// TwinCAT 3 PLC project TrafficPLC
// ProgramVersion: 3.1.4024.0
// libraries:
//   Tc2_Standard, * (Beckhoff Automation GmbH)
//   Tc2_System, * (Beckhoff Automation GmbH)
//   Tc3_Module, * (Beckhoff Automation GmbH)
// project tree:
//   / PlcTask.TcTTO
//   POUs/ MAIN.TcPOU
// real-time tasks:
//   TASK PlcTask: cycle T#10ms, priority 20, ADS port 350

CONFIGURATION TrafficPLC
    RESOURCE PLC ON TwinCAT3
        TASK PlcTask(INTERVAL := T#10ms, PRIORITY := 20);
        PROGRAM MAIN WITH PlcTask : MAIN;
    END_RESOURCE
END_CONFIGURATION

// ---- POUs/MAIN.TcPOU
PROGRAM MAIN
VAR
	//light states
	northIsRed : BOOL := TRUE; //Start of the program
	northIsYellow : BOOL := FALSE;
	northIsGreen : BOOL := FALSE;
	
	eastIsRed : BOOL := FALSE;
	eastIsYellow : BOOL := FALSE;
	eastIsGreen : BOOL := FALSE; 
	
	//timers
	northRedTimer: TON;
	northYellowTimer: TON;
	northGreenTimer: TON;
	
	eastRedTimer: TON;
	eastYellowTimer: TON;
	eastGreenTimer: TON;
	
	
	//amount of time each light stays on
	redTime : TIME := T#32S;  
	yellowTime : TIME := T#4S;
	greenTime : TIME := T#20S;
	
	
	//initial offset state
	isOffset : BOOL := TRUE; // Also starts the program off
	//offset timer and time value
	offsetTimer : TON;

	offsetTime : TIME := T#4S;
	
	
	
END_VAR

northRedTimer(IN := northIsRed, PT := redTime);
northYellowTimer(IN := northIsYellow, PT := yellowTime);
northGreenTimer(IN := northIsGreen, PT := greenTime);

eastRedTimer(IN := eastIsRed, PT := redTime);
eastYellowTimer(IN := eastIsYellow, PT := yellowTime);
eastGreenTimer(IN := eastIsGreen, PT := greenTime);


offsetTimer(IN:=isOffset, PT := offsetTime);


//Initial offset state
IF offsetTimer.Q THEN
	eastIsGreen := TRUE;
	isOffset := FALSE;
END_IF


//North Light Timings

IF northRedTimer.Q THEN
	northIsRed := FALSE;
	northIsGreen := TRUE;
END_IF

IF northGreenTimer.Q THEN
	northIsGreen := FALSE;
	northIsYellow := TRUE;
END_IF

IF northYellowTimer.Q THEN
	northIsYellow := FALSE;
	northIsRed := TRUE;
END_IF


//East Light Timings

IF eastRedTimer.Q THEN
	eastIsRed := FALSE;
	eastIsGreen := TRUE;
END_IF

IF eastGreenTimer.Q THEN
	eastIsGreen := FALSE;
	eastIsYellow := TRUE;
END_IF

IF eastYellowTimer.Q THEN
	eastIsYellow := FALSE;
	eastIsRed := TRUE;
END_IF

END_PROGRAM
